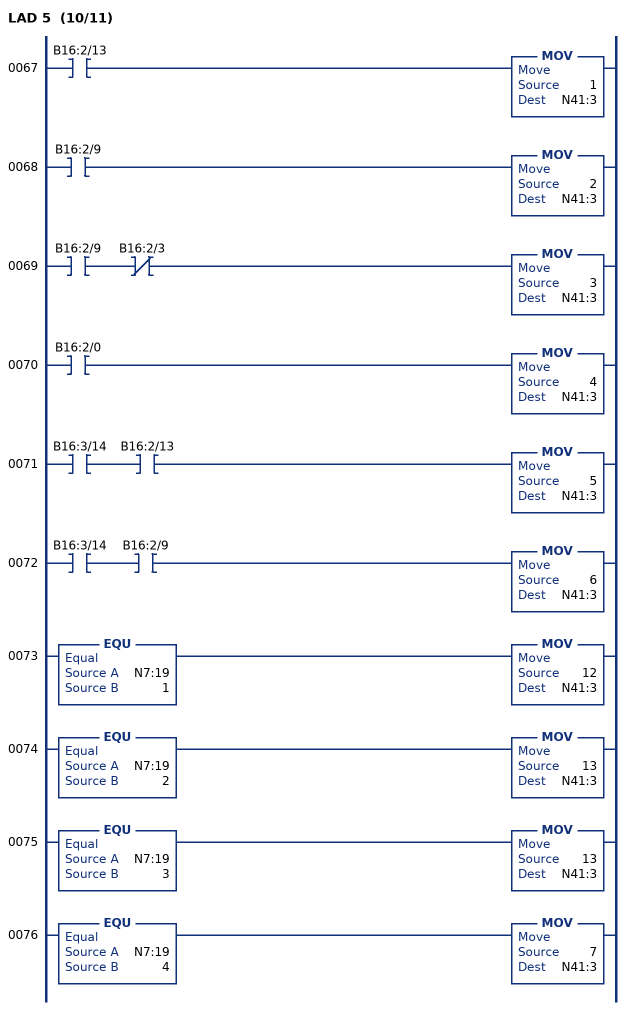
% Rung: 67 %
SOR XIC B16:2/13 MOV 1 N41:3 EOR
% Rung: 68 %
SOR XIC B16:2/9 MOV 2 N41:3 EOR
% Rung: 69 %
SOR XIC B16:2/9 XIO B16:2/3 MOV 3 N41:3 EOR
% Rung: 70 %
SOR XIC B16:2/0 MOV 4 N41:3 EOR
% Rung: 71 %
SOR XIC B16:3/14 XIC B16:2/13 MOV 5 N41:3 EOR
% Rung: 72 %
SOR XIC B16:3/14 XIC B16:2/9 MOV 6 N41:3 EOR
% Rung: 73 %
SOR EQU N7:19 1 MOV 12 N41:3 EOR
% Rung: 74 %
SOR EQU N7:19 2 MOV 13 N41:3 EOR
% Rung: 75 %
SOR EQU N7:19 3 MOV 13 N41:3 EOR
% Rung: 76 %
SOR EQU N7:19 4 MOV 7 N41:3 EOR

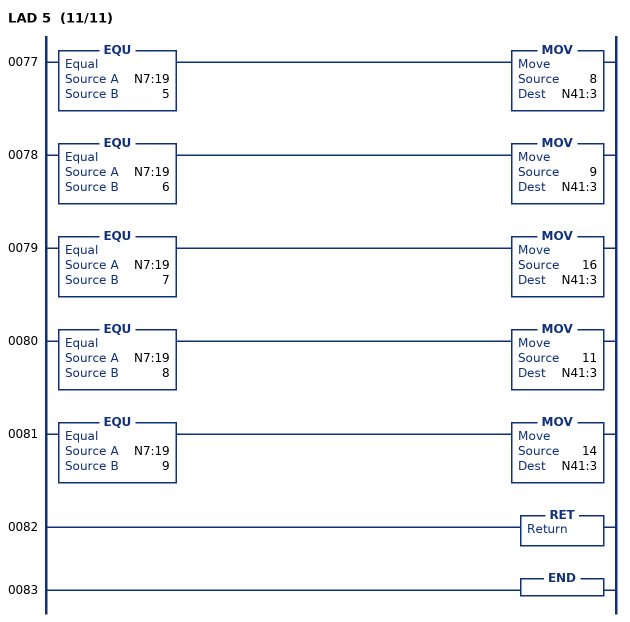
% Rung: 77 %
SOR EQU N7:19 5 MOV 8 N41:3 EOR
% Rung: 78 %
SOR EQU N7:19 6 MOV 9 N41:3 EOR
% Rung: 79 %
SOR EQU N7:19 7 MOV 16 N41:3 EOR
% Rung: 80 %
SOR EQU N7:19 8 MOV 11 N41:3 EOR
% Rung: 81 %
SOR EQU N7:19 9 MOV 14 N41:3 EOR
% Rung: 82 %
SOR RET EOR
% Rung: 83 %
SOR END EOR

LADDER 6
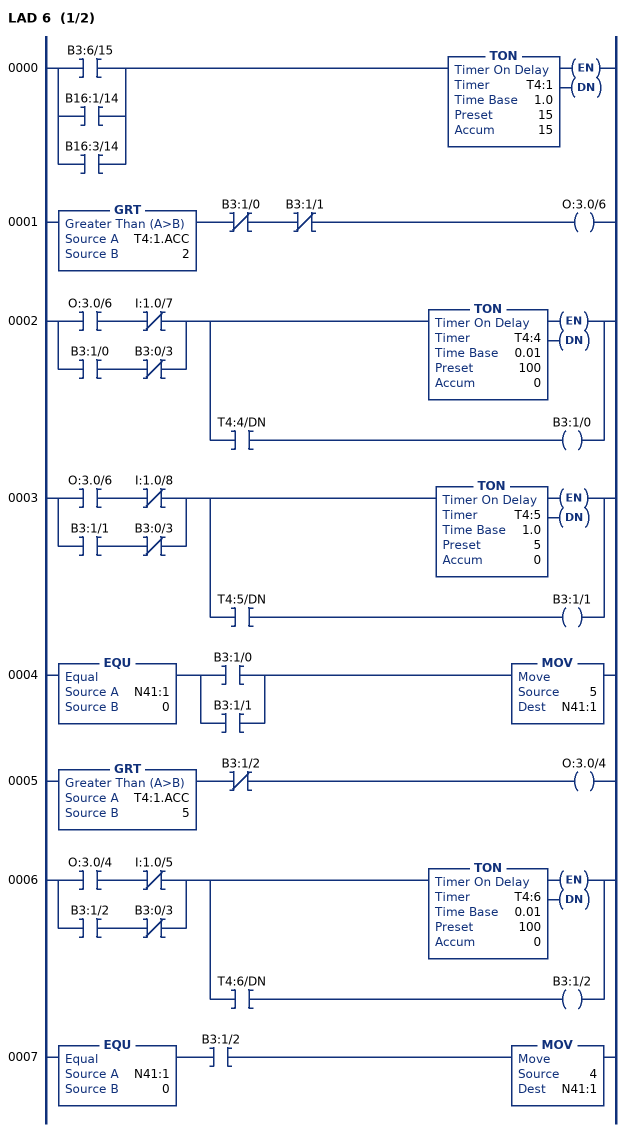
% Rung: 0 %
SOR BST XIC B3:6/15 NXB XIC B16:1/14 NXB XIC B16:3/14 BND TON T4:1 1.0 15 15 EOR
% Rung: 1 %
SOR GRT T4:1.ACC 2 XIO B3:1/0 XIO B3:1/1 OTE O:3.0/6 EOR
% Rung: 2 %
SOR BST XIC O:3.0/6 XIO I:1.0/7 NXB XIC B3:1/0 XIO B3:0/3 BND BST TON T4:4 0.01 100 0 NXB XIC T4:4/DN OTE B3:1/0 BND EOR
% Rung: 3 %
SOR BST XIC O:3.0/6 XIO I:1.0/8 NXB XIC B3:1/1 XIO B3:0/3 BND BST TON T4:5 1.0 5 0 NXB XIC T4:5/DN OTE B3:1/1 BND EOR
% Rung: 4 %
SOR EQU N41:1 0 BST XIC B3:1/0 NXB XIC B3:1/1 BND MOV 5 N41:1 EOR
% Rung: 5 %
SOR GRT T4:1.ACC 5 XIO B3:1/2 OTE O:3.0/4 EOR
% Rung: 6 %
SOR BST XIC O:3.0/4 XIO I:1.0/5 NXB XIC B3:1/2 XIO B3:0/3 BND BST TON T4:6 0.01 100 0 NXB XIC T4:6/DN OTE B3:1/2 BND EOR
% Rung: 7 %
SOR EQU N41:1 0 XIC B3:1/2 MOV 4 N41:1 EOR

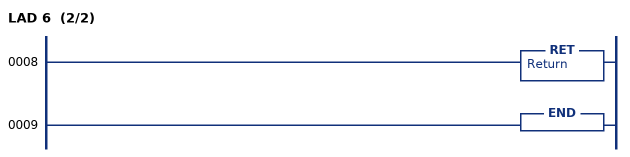
% Rung: 8 %
SOR RET EOR
% Rung: 9 %
SOR END EOR

LADDER 7
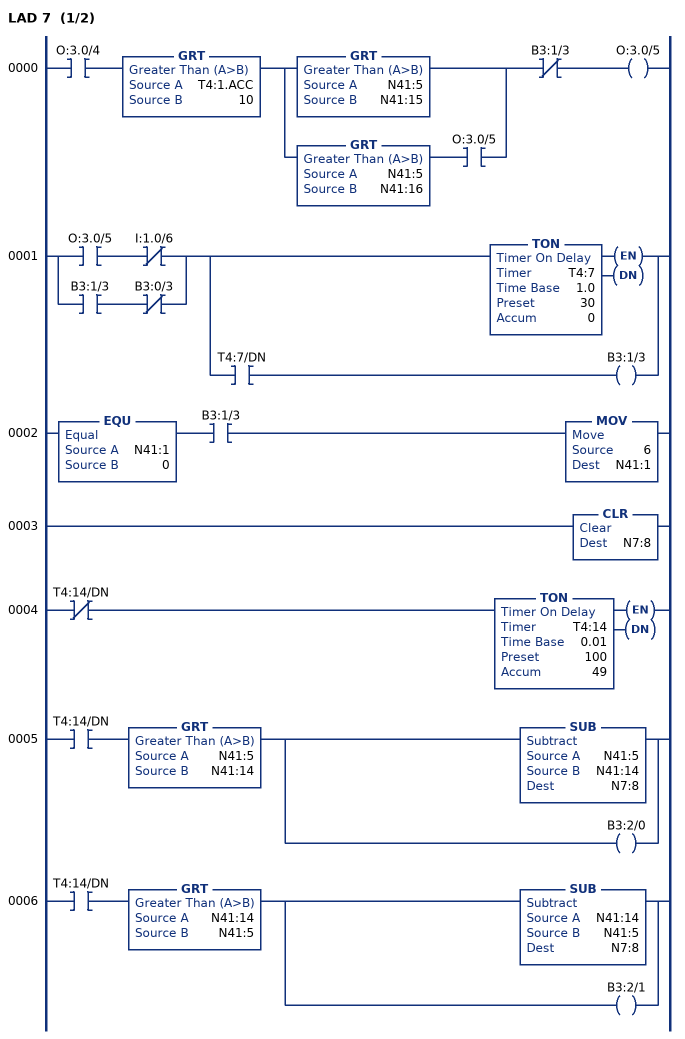
% Rung: 0 %
SOR XIC O:3.0/4 GRT T4:1.ACC 10 BST GRT N41:5 N41:15 NXB GRT N41:5 N41:16 XIC O:3.0/5 BND XIO B3:1/3 OTE O:3.0/5 EOR
% Rung: 1 %
SOR BST XIC O:3.0/5 XIO I:1.0/6 NXB XIC B3:1/3 XIO B3:0/3 BND BST TON T4:7 1.0 30 0 NXB XIC T4:7/DN OTE B3:1/3 BND EOR
% Rung: 2 %
SOR EQU N41:1 0 XIC B3:1/3 MOV 6 N41:1 EOR
% Rung: 3 %
SOR CLR N7:8 EOR
% Rung: 4 %
SOR XIO T4:14/DN TON T4:14 0.01 100 49 EOR
% Rung: 5 %
SOR XIC T4:14/DN GRT N41:5 N41:14 BST SUB N41:5 N41:14 N7:8 NXB OTE B3:2/0 BND EOR
% Rung: 6 %
SOR XIC T4:14/DN GRT N41:14 N41:5 BST SUB N41:14 N41:5 N7:8 NXB OTE B3:2/1 BND EOR

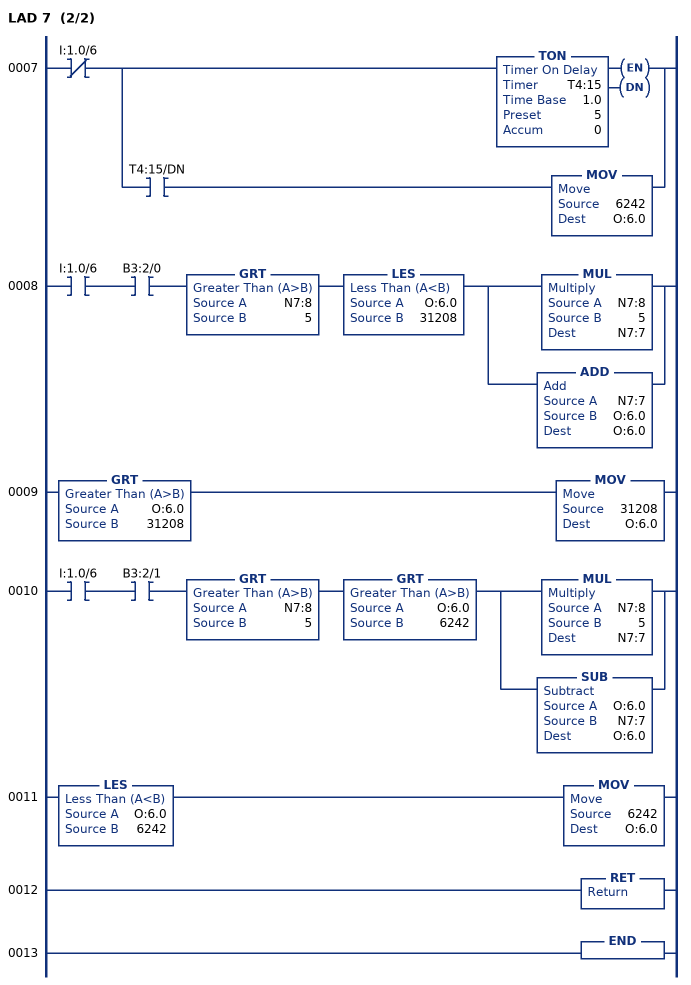
% Rung: 7 %
SOR XIO I:1.0/6 BST TON T4:15 1.0 5 0 NXB XIC T4:15/DN MOV 6242 O:6.0 BND EOR
% Rung: 8 %
SOR XIC I:1.0/6 XIC B3:2/0 GRT N7:8 5 LES O:6.0 31208 BST MUL N7:8 5 N7:7 NXB ADD N7:7 O:6.0 O:6.0 BND EOR
% Rung: 9 %
SOR GRT O:6.0 31208 MOV 31208 O:6.0 EOR
% Rung: 10 %
SOR XIC I:1.0/6 XIC B3:2/1 GRT N7:8 5 GRT O:6.0 6242 BST MUL N7:8 5 N7:7 NXB SUB O:6.0 N7:7 O:6.0 BND EOR
% Rung: 11 %
SOR LES O:6.0 6242 MOV 6242 O:6.0 EOR
% Rung: 12 %
SOR RET EOR
% Rung: 13 %
SOR END EOR

LADDER 8
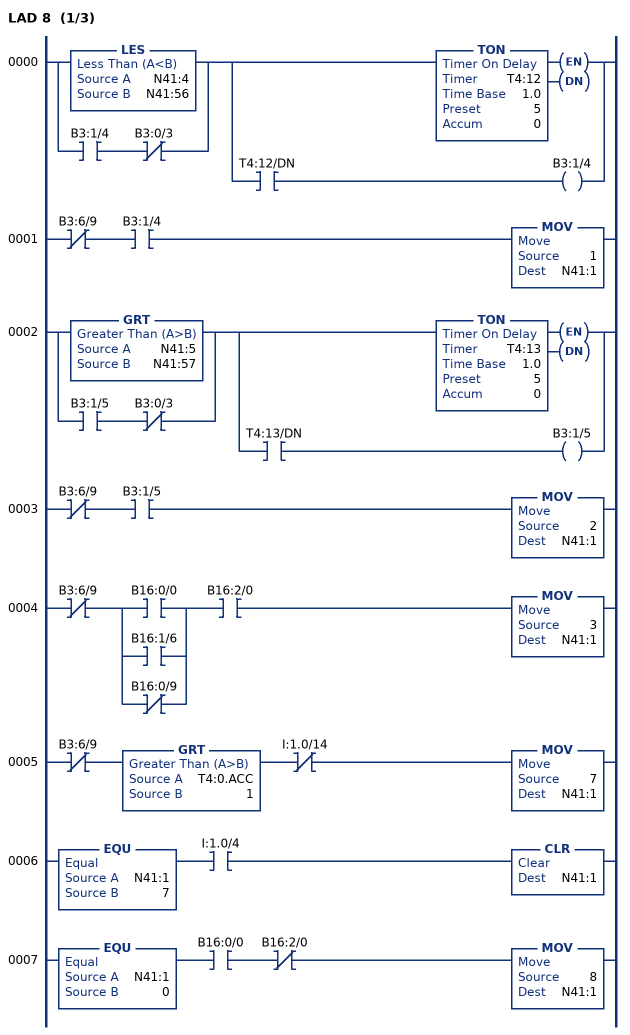
% Rung: 0 %
SOR BST LES N41:4 N41:56 NXB XIC B3:1/4 XIO B3:0/3 BND BST TON T4:12 1.0 5 0 NXB XIC T4:12/DN OTE B3:1/4 BND EOR
% Rung: 1 %
SOR XIO B3:6/9 XIC B3:1/4 MOV 1 N41:1 EOR
% Rung: 2 %
SOR BST GRT N41:5 N41:57 NXB XIC B3:1/5 XIO B3:0/3 BND BST TON T4:13 1.0 5 0 NXB XIC T4:13/DN OTE B3:1/5 BND EOR
% Rung: 3 %
SOR XIO B3:6/9 XIC B3:1/5 MOV 2 N41:1 EOR
% Rung: 4 %
SOR XIO B3:6/9 BST XIC B16:0/0 NXB XIC B16:1/6 NXB XIO B16:0/9 BND XIC B16:2/0 MOV 3 N41:1 EOR
% Rung: 5 %
SOR XIO B3:6/9 GRT T4:0.ACC 1 XIO I:1.0/14 MOV 7 N41:1 EOR
% Rung: 6 %
SOR EQU N41:1 7 XIC I:1.0/4 CLR N41:1 EOR
% Rung: 7 %
SOR EQU N41:1 0 XIC B16:0/0 XIO B16:2/0 MOV 8 N41:1 EOR

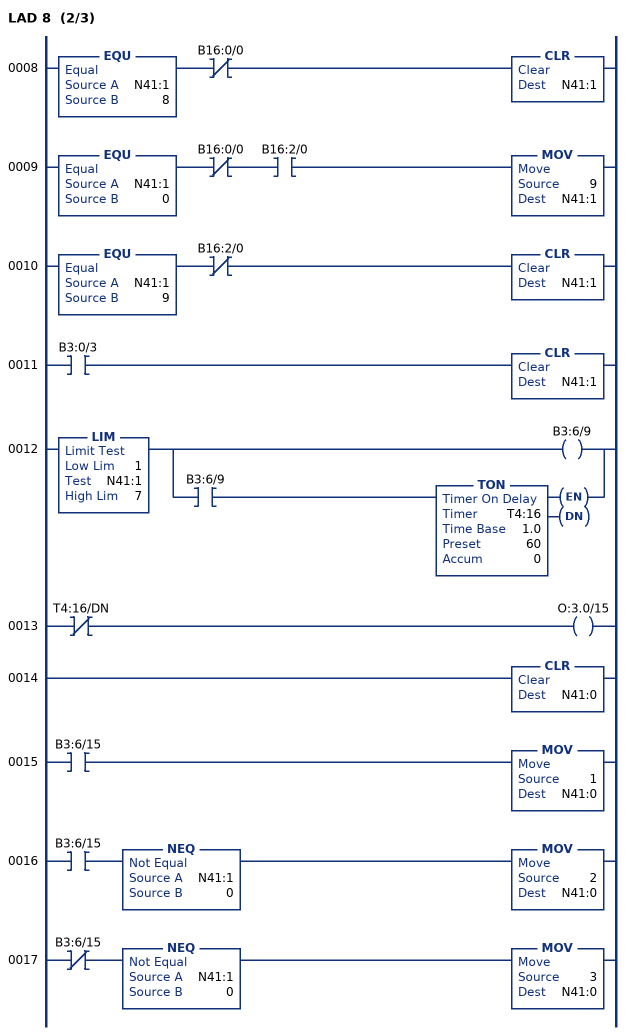
% Rung: 8 %
SOR EQU N41:1 8 XIO B16:0/0 CLR N41:1 EOR
% Rung: 9 %
SOR EQU N41:1 0 XIO B16:0/0 XIC B16:2/0 MOV 9 N41:1 EOR
% Rung: 10 %
SOR EQU N41:1 9 XIO B16:2/0 CLR N41:1 EOR
% Rung: 11 %
SOR XIC B3:0/3 CLR N41:1 EOR
% Rung: 12 %
SOR LIM 1 N41:1 7 BST OTE B3:6/9 NXB XIC B3:6/9 TON T4:16 1.0 60 0 BND EOR
% Rung: 13 %
SOR XIO T4:16/DN OTE O:3.0/15 EOR
% Rung: 14 %
SOR CLR N41:0 EOR
% Rung: 15 %
SOR XIC B3:6/15 MOV 1 N41:0 EOR
% Rung: 16 %
SOR XIC B3:6/15 NEQ N41:1 0 MOV 2 N41:0 EOR
% Rung: 17 %
SOR XIO B3:6/15 NEQ N41:1 0 MOV 3 N41:0 EOR

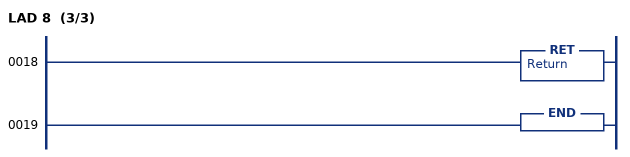
% Rung: 18 %
SOR RET EOR
% Rung: 19 %
SOR END EOR

DATA TABLE (non-zero values as saved)
DATA B3
% B3:0 % 0X0002 0X0000 0X0000 0X0000 0X0000 0X0000 0X8001 0X0000 0X0000 0X0000
DATA T4
% .PRE .ACC %
% T4:0 % 30 30
% T4:1 % 15 15
% T4:2 % 30 0
% T4:3 % 30 0
% T4:4 % 100 0
% T4:5 % 5 0
% T4:6 % 100 0
% T4:7 % 30 0
% T4:9 % 2 0
% T4:10 % 30000 0
% T4:11 % 30000 0
% T4:12 % 5 0
% T4:13 % 5 0
% T4:14 % 100 49
% T4:15 % 5 0
% T4:16 % 60 0
% T4:17 % 45 0
% T4:20 % 30000 30000
% T4:21 % 2000 2000
% T4:22 % 60 0
% T4:23 % 300 0
% T4:24 % 2000 2000
% T4:25 % 60 0
% T4:30 % 30000 0
% T4:31 % 2000 1160
% T4:32 % 60 0
% T4:33 % 300 0
% T4:34 % 2000 853
% T4:35 % 25 25
% T4:36 % 15 0
% T4:37 % 2000 0
% T4:38 % 2000 0
% T4:39 % 180 0
% T4:40 % 100 0
% T4:41 % 100 0
% T4:42 % 5 0
% T4:43 % 5 0
% T4:44 % 45 0
% T4:45 % 30 0
% T4:46 % 10 0
DATA N7
% N7:0 % 0 0 308 408 2 845 0 145 0 5
% N7:10 % 1 1 0 0 0 0 0 0 0 0
DATA B16
% B16:0 % 0X0A2A 0XD085 0X4000 0X2001 0X0000 0X0000 0X0000 0X0000 0X0000 0X0000
DATA N17
% N17:0 % 8192 2 10 10 137 0 0 224 5 142
% N17:10 % 0 20 3072 0 0 0 0 0 0 0
% N17:20 % 0 0 6 10 2 0 0 0 0 0
DATA N18
% N18:0 % 8192 2 10 11 137 0 0 224 5 143
% N18:10 % 0 20 3072 0 0 0 0 0 0 0
% N18:20 % 0 1 0 0 0 0 0 0 0 0
DATA B40
% B40:0 % 0X0000 0X0000 0X0000 0X0000 0X0000 0X0000 0X0001 0X0082 0X0000 0X0000
DATA N41
% N41:0 % 1 0 6 0 35 881 1 2 0 0
% N41:10 % 35 10 30 10 850 900 820 0 0 0
% N41:20 % 50 10 200 60 500 5 500 500 0 0
% N41:30 % 100 10 300 110 200 20 800 220 0 0
% N41:40 % 1200 60 1200 50 1200 1230 0 0 0 0
% N41:50 % 45 33 834 0 2 526 -40 1450 0 0
% N41:60 % 92 75 100 -50 1400 0 0 0 0 0
DATA B42
% B42:0 % 0X0080 0X0000 0X0000 0X0000 0X0000 0X0000 0X0000 0X0000 0X0000 0X0000
